{attribute addProperty BoxType "EL1502-0000-0018"}
{attribute addProperty Id "ControlAT %Q*Control_1E8AA4851621Set_counter_valueAT %Q*UDINT32417"}
{attribute addProperty CRC "186355450"}
{attribute addProperty SizeInBites "48"}
{attribute addProperty SizeInBytes "6"}
TYPE CNT_Outputs_0B1B8EFA :
STRUCT
	{attribute addProperty Name "Control"}
	Control AT %Q* : Control_1E8AA485;
	{attribute addProperty Name "Set_counter_value"}
	Set_counter_value AT %Q* : UDINT;
END_STRUCT
END_TYPE

(* stored: Version 1.2.0.0, ProductVersion 3.1.4024.9
   DUT CNT_Outputs_0B1B8EFA: Id {e45b5023-c4df-4ab8-9dc5-39bf91f46d1f} *)
